// TwinCAT 3 PLC project Automation_App
// ProgramVersion: 3.1.4026.21
// libraries:
//   Tc2_MC2, * (Beckhoff Automation GmbH)
//   Tc2_Standard, * (Beckhoff Automation GmbH)
//   Tc2_System, * (Beckhoff Automation GmbH)
//   Tc2_Utilities, * (Beckhoff Automation GmbH)
//   Tc3_Module, * (Beckhoff Automation GmbH)
//   BASIC,3.31,OSCAT
// project tree:
//   GVLs/ GVL_VFD.TcGVL
//   / PlcTask.TcTTO
//   POUs/InputConveyor/ FB_InputConvBufferManagement.TcPOU, FB_InputConvVFD.TcPOU, FB_InputConvProperties.TcPOU, FB_InputConvMAIN.TcPOU, ST_InputConvData.TcDUT
//   POUs/ MAIN.TcPOU
//   POUs/OutputConveyor/ FB_OutputConvVFD.TcPOU, ST_OutputConvData.TcDUT, FB_OutputConvBufferManagement.TcPOU, FB_OutputConvMain.TcPOU, FB_OutputConvProperties.TcPOU
//   POUs/RobotInterface/ FB_RobotInterefaceMAIN.TcPOU
// real-time tasks:
//   TASK PlcTask: cycle T#1ms, priority 20, ADS port 350

CONFIGURATION Automation_App
    RESOURCE PLC ON TwinCAT3
        TASK PlcTask(INTERVAL := T#1ms, PRIORITY := 20);
        PROGRAM MAIN WITH PlcTask : MAIN;
    END_RESOURCE
END_CONFIGURATION

// ---- POUs/InputConveyor/ST_InputConvData.TcDUT
TYPE ST_InputConvData :
STRUCT
	id :INT; // Unique box identifier assigned on entry
	timeStampin :STRING; // Timestamp when box passed the entry (IN) sensor
	timeStamparrived:STRING; // Timestamp when box reached the exit (OUT) sensor
	timeStampout:STRING; // Timestamp when box cleared the exit (OUT) sensor
END_STRUCT
END_TYPE

// ---- POUs/OutputConveyor/ST_OutputConvData.TcDUT
TYPE ST_OutputConvData :
STRUCT
	id :INT; // Unique box identifier assigned when robot places the box
	timeStampin :STRING; // Timestamp when box entered the drop zone (IN sensor rising edge)
	timeStampout:STRING; // Timestamp when box left the conveyor (OUT sensor falling edge)
END_STRUCT
END_TYPE

// ---- GVLs/GVL_VFD.TcGVL
{attribute 'qualified_only'}
VAR_GLOBAL
	
// INPUT Conveyor----------------------
// Outputs from PLC to input conveyor VFD
	bInConvStop			AT%Q*:BOOL; // Stop command to input conveyor VFD
    bInConvRunFWD		AT%Q*:BOOL; // Run forward command to input conveyor VFD
	bInConvRunREV		AT%Q*:BOOL; // Run reverse command to input conveyor VFD
	bInConvJog			AT%Q*:BOOL; // Jog command to input conveyor VFD

// Inputs from input conveyor VFD to PLC
	bInputVFDSpeedReached	AT%I*:BOOL; // Speed-reached status from input conveyor VFD
	bInConvFault			AT%I*:BOOL; // Fault status from input conveyor VFD
	bInputVFDRunning		AT%I*:BOOL; // Running status from input conveyor VFD
	
// Inputs form Conveyor Sensors
	bInputConveyorINSensor	AT%I*:BOOL; // Entry photo sensor on input conveyor (box arriving)
	bInputConveyorOUTSensor AT%I*:BOOL; // Exit photo sensor on input conveyor (box at robot pickup position)

// OUTPUT CONVEYOR-----------------------
// Outputs from PLC to input conveyor VFD
	bOutConvStop		AT%Q*:BOOL; // Stop command to output conveyor VFD
    bOutConvRunFWD		AT%Q*:BOOL; // Run forward command to output conveyor VFD
	bOutConvRunREV		AT%Q*:BOOL; // Run reverse command to output conveyor VFD
	bOutConvJog			AT%Q*:BOOL; // Jog command to output conveyor VFD

// Inputs from input conveyor VFD to PLC
	bOutputVFDSpeedReached	AT%I*:BOOL; // Speed-reached status from output conveyor VFD
	bOutConvFault			AT%I*:BOOL; // Fault status from output conveyor VFD
	bOutputVFDRunning		AT%I*:BOOL; // Running status from output conveyor VFD
	
// Inputs form Conveyor Sensors
	bOutputConveyorINSensor		AT%I*:BOOL; // Entry photo sensor on output conveyor (robot drop zone)
	bOutputConveyorOUTSensor	AT%I*:BOOL; // Exit photo sensor on output conveyor (box leaving system)
END_VAR

// ---- POUs/MAIN.TcPOU
PROGRAM MAIN
VAR
    InputConveyor	:FB_InputConvMAIN;      // Input conveyor subsystem controller
	RobotInterface	:FB_RobotInterefaceMAIN; // Robot pick/place coordination
	OutputConveyor	:FB_OutputConvMAIN;     // Output conveyor subsystem controller

    bEnable		:BOOL; //PLC Logic Enable
	bInFeedtoConv :BOOL:= TRUE; // Allow external infeed system to feed boxes onto input conveyor
	rCyclePLC	:REAL:= 0.001; // PLC task cycle time in seconds (1 ms default)
	bSimulation :BOOL; // TRUE = run in simulation mode (no real hardware required)
	
END_VAR

InputConveyor(
	bEnable:= bEnable , 
	bInFeedtoConv:= bInFeedtoConv , 
	bRobotReadytoPick:= RobotInterface.bRobotReadyPickInputConv , 
	rCyclePLC:= rCyclePLC, 
	bSimulation:= bSimulation, 
	AllowInFeedtoInputConv=> , 
	AllowOutFeedtoRobot=> );

//RobotInterface
RobotInterface(
	bEnable := bEnable,
	bInputConvReady:= InputConveyor.AllowOutFeedtoRobot ,
	bOutputConvReady:= outputconveyor.AllowRobotPlace ,
	bRobotReadyPickInputConv=> ,
	bRobotReadyPlaceOutputConv=> );

//InputConveyor(
OutputConveyor(
	bEnable:= bEnable , 
	bRobotReadytoPlace:= RobotInterface.bRobotReadyPlaceOutputConv , 
	rCyclePLC:= rCyclePLC , 
	bSimulation:= bSimulation, 
	AllowRobotPlace=>);

END_PROGRAM

// ---- POUs/InputConveyor/FB_InputConvMAIN.TcPOU
FUNCTION_BLOCK FB_InputConvMAIN
VAR_INPUT
	bEnable			:BOOL; //PLC Logic Enable
	bInFeedtoConv 	:BOOL; //Outside signal from infeed system to conveyor - ready to recieve
	bRobotReadytoPick 	:BOOL; //Outside signal from robot - ready to recieve
	rCyclePLC			:REAL; // PLC task cycle time in seconds
	bSimulation :BOOL; // TRUE = VFD simulation active (no real drive)
	
END_VAR
VAR_OUTPUT
	AllowInFeedtoInputConv :BOOL; //Allow infeed of new boxes signal
	AllowOutFeedtoRobot :BOOL; //Ready to be picked up by robot signal
END_VAR
VAR
	//Function Blocks
	InputConvPropeties		:FB_InputConvProperties;
	InputConvVFD			:FB_InputConvVFD;
	InputConvBufferManger	:FB_InputConvBufferManagement;

	iMotorMaxSpeed			:INT; // Motor rated speed at 50 Hz [RPM]
	iConveyorVelocitycmd	:REAL; // Commanded belt velocity [m/s]
	rAccTime				:REAL; // Drive acceleration time [s]
	rDecTime				:REAL; // Drive deceleration time [s]

	//Belt linear vel tranformation
	iGearboxReduction	:INT := 1; // Gearbox reduction ratio (motor to pulley shaft)
	rPullyDiameter		:REAL; // Drive pulley diameter [m]
	
	//Conveyor propeties 
	rConvLength :REAL; //Conveyor Length in m (Distance between sensors)
	rBoxLen	:REAL; //Box size length in m
	rMinGap	:REAL; //Allowable min gap between boxes in m
	
END_VAR



InputConvBufferManger(
	bEnable:= bEnable , 
	bInSensor:= GVL_VFD.bInputConveyorINSensor, 
	bOutSensor:= GVL_VFD.bInputConveyorOUTSensor ,
	bReadytoRecieve:= bInFeedtoConv, 
	rConvLength:= rConvLength , 
	rBoxLen:= rBoxLen , 
	rMinGap:= rMinGap , 
	bRobotReady:= bRobotReadytoPick);

AllowInFeedtoInputConv := InputConvBufferManger.bAllowIn;
AllowOutFeedtoRobot := InputConvBufferManger.bAllowOut;
	
InputConvPropeties(
	GearboxReduction:= iGearboxReduction , 
	PullyDiameter:= rPullyDiameter , 
	ConveyorVelocitycmd:= iConveyorVelocitycmd  , 
	MotorMaxSpeed:= iMotorMaxSpeed,
	bBufferFull:= InputConvBufferManger.bFull);

IF bSimulation THEN 

	InputConvVFD(
		bStop:= GVL_VFD.bInConvStop, 
		bRunFWR:= GVL_VFD.bInConvRunFWD, 
		bRunREV:= GVL_VFD.bInConvRunREV , 
		bJog:= GVL_VFD.bInConvJog , 
		iVoltage:= InputConvPropeties.AnalogOut_V,
		iVoltageMax:= 10,
		rAccTime:= rAccTime , 
		rDecTime:= rDecTime,
		iMotorMaxSpeed:= iMotorMaxSpeed,
		ConveyorVelocityMax:= InputConvPropeties.ConveyorVelocityMax);
		
END_IF

GVL_VFD.bInputVFDSpeedReached	:= InputConvVFD.bSpeedReached;
GVL_VFD.bInputVFDRunning		:= InputConvVFD.bRunning;
//GVL_VFD.bInConvFault	:= ;

END_FUNCTION_BLOCK

// ---- POUs/InputConveyor/FB_InputConvProperties.TcPOU
FUNCTION_BLOCK FB_InputConvProperties
VAR_INPUT 
	bEnable				:BOOL; // PLC Logic Enable
	GearboxReduction 	:INT; // Gearbox reduction ratio (motor to pulley shaft)
	PullyDiameter		:REAL; //m
	ConveyorVelocitycmd	:REAL; //m/s
	MotorMaxSpeed		:INT; //RPM at 50 Hz (ASSUMPTION)
	bBufferFull			:BOOL; // Forces motor speed to zero when the conveyor buffer is full
	
END_VAR

VAR_OUTPUT
	ConveyorVelocityMax  :REAL; // [m/s] at MotorMaxSpeed
    MotorRPM             :REAL; // [rpm]
    MotorHz              :REAL; // [Hz] 0..50
    AnalogOut_V          :REAL; // [V] 0..10
    AnalogOut_Raw     AT%Q*: INT;   // 0..32767
END_VAR

VAR
	HzMax 	:REAL :=50; // Maximum drive frequency [Hz]
    HzCmd	:REAL; // Calculated frequency command [Hz]
    Vin		:REAL; // Calculated analog output voltage [V]
    RawAnalog	:REAL; // Intermediate raw analog value before INT conversion
END_VAR

IF PullyDiameter = 0.0 OR MotorMaxSpeed = 0 OR GearboxReduction = 0 THEN
	ConveyorVelocityMax := 0;
ELSE
	ConveyorVelocityMax := (PullyDiameter*PI*(MotorMaxSpeed/GearboxReduction))/60; // m/s
END_IF

IF bBufferFull THEN
    MotorRPM := 0.0;	// forced stop
ELSIF (PullyDiameter > 0.0) AND (GearboxReduction > 0.0) THEN
    MotorRPM := (ConveyorVelocitycmd * 60.0 * GearboxReduction) / (LREAL_TO_REAL (PI) * PullyDiameter);	// RPM
ELSE
    MotorRPM := 0.0;	// invalid mechanics
END_IF;

// RPM -> Hz (0..50)
IF (MotorMaxSpeed <= 0.0) THEN
	HzCmd := 0.0;
ELSE
	HzCmd := (MotorRPM / MotorMaxSpeed) * HzMax;
END_IF

// Clamp Hz to 0..50
IF HzCmd < 0.0 THEN
	HzCmd := 0.0;
ELSIF HzCmd > HzMax THEN
	HzCmd := HzMax;
END_IF
MotorHz := HzCmd;

// Hz -> 0..10V (linear)
Vin := (HzCmd / HzMax) * 10.0;

// Clamp V to 0..10
IF Vin < 0.0 THEN
	Vin := 0.0;
ELSIF Vin > 10.0 THEN
	Vin := 10.0;
END_IF
AnalogOut_V := Vin;

// 0..10V -> 0..32767 counts
RawAnalog := (Vin / 10.0) * 32767.0;

// Clamp counts
IF RawAnalog < 0.0 THEN
	RawAnalog := 0.0;
ELSIF RawAnalog > 32767.0 THEN
	RawAnalog := 32767.0;
END_IF

AnalogOut_Raw := REAL_TO_INT(LREAL_TO_REAL(RawAnalog));

END_FUNCTION_BLOCK

// ---- POUs/InputConveyor/FB_InputConvVFD.TcPOU
//Generate commands to a drive.
FUNCTION_BLOCK FB_InputConvVFD

VAR_INPUT
	bStop				:BOOL; // Stop command - resets SRAMP and forces velocity to zero
    bRunFWR				:BOOL; // Run forward command
	bRunREV				:BOOL; // Run reverse command
	bJog		:BOOL; // Jog command (treated the same as forward run)
	iVoltage		:REAL; // Analog speed reference voltage [V]
	iVoltageMax		:REAL; // Maximum analog reference voltage [V] (typically 10 V)
    rAccTime		:REAL;      // Acc in seconds
    rDecTime		:REAL;      // DEC in seconds
	iMotorMaxSpeed	:REAL; // Motor rated speed at 50 Hz [RPM]
	ConveyorVelocityMax :REAL; // Maximum conveyor belt velocity at motor max speed [m/s]
	
END_VAR

VAR_OUTPUT
	bSpeedReached	:BOOL; // TRUE when drive output frequency matches the reference
	bFault			:BOOL; // Drive fault flag (not implemented in simulation)
	bRunning		:BOOL; // TRUE when drive is running with a positive frequency reference
	rDriveVelProfile	:REAL;   // Simulated Motor vel profile
	rDriveACCProfile	:REAL; // Simulated Motor acc profile
	
END_VAR

VAR
	DriveRun		:BOOL; // TRUE when exactly one direction command is active (XOR result)
    DriveRunFWR		:BOOL; // Internal forward run (RunFWR OR Jog)
    DriveRunREV		:BOOL; // Internal reverse run
    DriveHzRef		:REAL; // Target frequency reference [Hz], ±HzMax
	rAccRate		:REAL; // Acceleration rate [Hz/s]
    rDecRate		:REAL; // Deceleration rate [Hz/s] (negative value)
	rDirSign 		:REAL; // Direction sign: +1.0 forward, -1.0 reverse
	fbSRAMP :SRAMP; // OSCAT S-ramp function block for smooth velocity profiling
	HzMax :REAL := 50; // Maximum drive frequency [Hz]
	rRPMvel :REAL; // Simulated motor shaft speed [RPM]
	rLinearVel :REAL; // Simulated conveyor belt linear velocity [m/s]
	sStatus		:STRING(120);	// STATUS text

END_VAR

// Run command
DriveRunFWR := bRunFWR OR bJog;
DriveRunREV := bRunREV;

DriveRun := (DriveRunFWR XOR DriveRunREV);   // TRUE only if one is on

IF bRunFWR OR bJog THEN
    rDirSign := 1.0;
ELSIF bRunREV THEN
    rDirSign := -1.0;

END_IF;

//Voltage to Hz:
IF iVoltage <= 0.0  THEN //OR NOT DriveRun
    DriveHzRef := 0.0;
ELSIF iVoltage > iVoltageMax THEN
    DriveHzRef := HzMax;
ELSE
    DriveHzRef := (iVoltage / iVoltageMax) * HzMax;
END_IF;


IF ABS(DriveHzRef) < 0.001 AND rAccTime > 0 THEN
    rAccRate := (HzMax / 2) / rAccTime;
ELSIF rAccTime > 0.01 THEN
    rAccRate := DriveHzRef / rAccTime;
ELSE
    rAccRate := DriveHzRef * 10.0;
END_IF;

IF ABS(DriveHzRef) < 0.001 AND rDecTime > 0 THEN
    rDecRate := (HzMax / 2) / -rDecTime;
ELSIF rDecTime > 0.01 THEN
	rDecRate := DriveHzRef / -rDecTime;   // Hz/s
ELSE
	rDecRate := DriveHzRef * -10.0;      // Hz/s
END_IF;

// Determine target input
IF DriveRun THEN 
	DriveHzRef := DriveHzRef * rDirSign;
ELSE
	DriveHzRef := 0.0;
END_IF;

// SRAMP function to build velocity command
fbSRAMP(
    X           := DriveHzRef,
    A_UP        := rAccRate,
    A_DN        := rDecRate,
    VU_MAX      := rAccRate *1000,     // Jerk
    VD_MAX      := rDecRate *1000,     // Jerk
    LIMIT_HIGH  := HzMax,
    LIMIT_LOW   := -HzMax,
    RST         := bStop ,
    Y           => rDriveVelProfile,
    V           => rDriveACCProfile // Acctual Acc
);

rRPMvel := rDriveVelProfile/HzMax * iMotorMaxSpeed;
rLinearVel := rDriveVelProfile/HzMax * ConveyorVelocityMax;

//Status
bSpeedReached := (rDriveVelProfile = DriveHzRef AND DriveRun );
bRunning      := (DriveHzRef > 0 AND DriveRun);

//Drive Status (priority-based)
IF bStop THEN
    // SRAMP reset → forced stop
    sStatus := 'STOP';

ELSIF (DriveRunFWR AND DriveRunREV) THEN
    // Illegal command combination
    sStatus := 'Command Conflict: Run Farward and Reverse';

ELSIF NOT DriveRun THEN
    // No valid run command (XOR result = FALSE)
    sStatus := 'Stopped (No specific direction Run Command)';

ELSE
    // DriveRun = TRUE (exactly one direction active)

    IF bRunFWR OR bJog THEN
        sStatus := 'Running Farward';

    ELSIF bRunREV THEN
        sStatus := 'Running Reverse';

    END_IF
END_IF;

END_FUNCTION_BLOCK

// ---- POUs/InputConveyor/FB_InputConvBufferManagement.TcPOU
FUNCTION_BLOCK FB_InputConvBufferManagement
VAR_INPUT

	bEnable	:BOOL; // PLC Logic Enable
    bInSensor	:BOOL; // Photo sensors
    bOutSensor	:BOOL; // Photo sensors
	bReadytoRecieve	:BOOL; //Ready to recieve from Robot
	// iCapacity	:INT; // For real system 
	
	// Geometry 
    rConvLength	:REAL;	// usable buffer length for simulation (meters)
    rBoxLen		:REAL;	// box length along travel for simulation (meters)
    rMinGap		:REAL;	// minimum clear gap between boxes for simulation (meters)
	
	bInfeedReady :BOOL:= TRUE; // Infeed Handshake
    bRobotReady	:BOOL:= TRUE; // Robot Handshake

END_VAR

VAR CONSTANT
    iMax_Boxes_buffer	:INT := 500; //  Expected max capacity FIFO storage size
END_VAR

VAR_OUTPUT
    bFull		:BOOL;			// Buffer is full (box count >= effective capacity)
    bEmpty		:BOOL;			// Buffer is empty (no boxes on conveyor)
    bAllowIn	:BOOL;			//Allow infeeder 
    bAllowOut	:BOOL;			//Allow Robot Pick
	
END_VAR

VAR
	bEnableBuffer :BOOL; // Enables FIFO tracking (must be TRUE for box counting to run)
		
    rtIn		:R_TRIG;	// Rising edge detector for bInSensor
    rtOut		:R_TRIG;	// Rising edge detector for bOutSensor
	ftOutOff	:F_TRIG;	// falling edge detector for bOutSensor
	
	bReset		:BOOL := FALSE; // Reset count on rising edge
    rtReset		:R_TRIG;	// Ralling edge reset
	
	iCount       :INT;     // current box count
    bInEdge      :BOOL;    // IN rising edge
    bOutEdge     :BOOL;    // OUT rising edge
	
	// Time
    fbTime	:FB_LocalSystemTime := (bEnable := TRUE, dwCycle := 1); // Local system time FB for box timestamping
    sNow	:STRING; // Current timestamp as formatted string
	
	//stData : ST_Data;
	Inputlog     : ARRAY[1..iMax_Boxes_buffer] OF ST_InputConvData; // FIFO array storing box tracking records
	
	// FIFO storage
    iHead	:INT := 1; // Index of the oldest box (next to dequeue)
    iTail	:INT := 1; // Index of the next empty slot (where next box is enqueued)
    iQCount	:INT := 0; // Current number of boxes in the FIFO

	// ID generator
    iIdCounter : INT := 0; // Auto-incrementing box ID counter (wraps at 32767)

	// Effective capacity
    iEffCap  : INT; // Effective buffer capacity after clamping (>= 0)

	iCapacity	:INT; // Configured maximum number of boxes on conveyor
	// Capacity intermediates
    rPitch_m	:REAL; // Box pitch = box length + minimum gap [m]
    rCap		:REAL; // Float capacity before floor truncation
    iCapTmp		:INT; // Intermediate capacity before final clamping

	i :INT; // Loop index used during FIFO reset
	sStatus		:STRING(120);	// STATUS text
END_VAR

//Capacity calculation -  For simulation
// IF (rBoxLen <= 0.0) OR (rMinGap <= 0.0) OR (rConvLength <= 0.0) THEN
//     iCapTmp := 0;
// ELSE
//     rPitch_m := rBoxLen + rMinGap;
// 
//     IF rPitch_m <= 0.0 THEN
//         iCapTmp := 0;
//     ELSE
//         rCap := (rConvLength + rMinGap) / rPitch_m;
// 
//         // Round down
//         iCapTmp := REAL_TO_INT(FLOOR(rCap));
// 
//         IF iCapTmp < 0 THEN
// 			iCapTmp := 0; 
// 		END_IF
//     END_IF
// END_IF
// 
// iCapacity := iCapTmp;

// Clamp to FIFO storage
iEffCap := iCapacity;

IF iEffCap < 0 THEN
	iEffCap := 0;
END_IF

//Timestamps
fbTime();
IF fbTime.bValid THEN
    sNow := SYSTEMTIME_TO_STRING(fbTime.systemTime);
ELSE
    sNow := '';
END_IF

// Edge detection
rtIn(CLK := bInSensor);
rtOut(CLK := bOutSensor);
rtReset(CLK := bReset);
ftOutOff(CLK := bOutSensor);

bInEdge  := rtIn.Q;
bOutEdge := rtOut.Q;

//Reset
IF rtReset.Q THEN
	
    iHead := 1;
    iTail := 1;
    iQCount := 0;
	
    FOR i := 1 TO iMax_Boxes_buffer DO
        Inputlog[i].id := 0;
        Inputlog[i].timeStampIn := '';
        Inputlog[i].timeStampArrived := '';
        Inputlog[i].timeStampOut := '';
    END_FOR

END_IF
	
//FIFO tracking
IF bEnable AND bEnableBuffer AND fbTime.bValid THEN

    // 1) IN rising edge > Push (if not full)
    IF bInEdge THEN
        IF iQCount < iEffCap THEN

            // ID wrap protection
            IF iIdCounter >= 32767 THEN
				iIdCounter := 0; 
			END_IF
            iIdCounter := iIdCounter + 1;

            Inputlog[iTail].id := iIdCounter;
            Inputlog[iTail].timeStampIn := sNow;
            Inputlog[iTail].timeStampArrived := '';
            Inputlog[iTail].timeStampOut := '';

            // advance tail
            iTail := iTail + 1;
            IF iTail > iMax_Boxes_buffer THEN
				iTail := 1;
			END_IF

            iQCount := iQCount + 1;
        END_IF
    END_IF


    // 2) OUT rising edge > stamp ARRIVED on oldest (HEAD)
    IF bOutEdge THEN
        IF iQCount > 0 THEN
            Inputlog[iHead].timeStampArrived := sNow;
        END_IF
    END_IF


    // 3) OUT falling edge -> stamp OUT on oldest and POP
    IF ftOutOff.Q THEN
        IF iQCount > 0 THEN
            Inputlog[iHead].timeStampOut := sNow;

            // pop
            iHead := iHead + 1;
            IF iHead > iMax_Boxes_buffer THEN
				iHead := 1;
			END_IF

            iQCount := iQCount - 1;
        END_IF
    END_IF

END_IF


iCount := iQCount; //Number of boxes on conveyor
bEmpty := (iCount <= 0);
bFull  := (iEffCap > 0) AND (iCount >= iEffCap);

// Send infeeder allow signal
bAllowIn  := bEnable AND NOT bFull AND NOT bInSensor AND bInfeedReady AND bReadytoRecieve;

// Outfeed release allowed if buffer has boxes AND robot is ready AND out sensor is blocked
bAllowOut := bEnable AND NOT bEmpty AND bOutSensor AND bRobotReady;

// Status (priority-based)
IF NOT bEnable THEN
    sStatus := 'Input-Conveyor Buffer - Disabled';

	// Hard limit states
	ELSIF bFull THEN
		sStatus := 'Conveyor is Full: STOP';
	ELSIF bEmpty THEN
		sStatus := 'Conveyor is Empty';

	// Infeed path (not full, not empty)
	ELSIF NOT bAllowIn THEN
		// Give the most relevant reason
		IF bInSensor THEN
			sStatus := 'Infeed blocked: entry sensor occupied';
		ELSIF NOT bInfeedReady THEN
			sStatus := 'Infeed blocked: infeeder not ready';
		ELSIF NOT bReadytoRecieve THEN
			sStatus := 'Infeed blocked: buffer not ready to receive';
		ELSE
			sStatus := 'Infeed blocked';
		END_IF

	// Outfeed path
	ELSIF NOT bAllowOut THEN
		IF NOT bOutSensor THEN
			sStatus := 'Outfeed waiting: no box at out sensor';
		ELSIF NOT bRobotReady THEN
			sStatus := 'Outfeed waiting: robot not ready';
		ELSE
			sStatus := 'Outfeed blocked';
		END_IF
ELSE
    sStatus := 'Running: Infeed/Outfeed allowed';
END_IF

END_FUNCTION_BLOCK

// ---- POUs/RobotInterface/FB_RobotInterefaceMAIN.TcPOU
FUNCTION_BLOCK FB_RobotInterefaceMAIN
VAR_INPUT
	bEnable :BOOL; // PLC Logic Enable
	bInputConvReady :BOOL; // Signal from input conveyor: box is ready at robot pickup position
	bOutputConvReady :BOOL; // Signal from output conveyor: drop zone is clear
	
END_VAR

VAR_OUTPUT
	bRobotReadyPickInputConv :BOOL; // Permission to robot: OK to pick from input conveyor
	bRobotReadyPlaceOutputConv :BOOL; // Permission to robot: OK to place on output conveyor
	
END_VAR
VAR
	
END_VAR

IF bEnable THEN
	bRobotReadyPickInputConv := TRUE;
	bRobotReadyPlaceOutputConv := TRUE;
ELSE
	bRobotReadyPickInputConv := FALSE;
	bRobotReadyPlaceOutputConv := FALSE;
END_IF

END_FUNCTION_BLOCK

// ---- POUs/OutputConveyor/FB_OutputConvMain.TcPOU
FUNCTION_BLOCK FB_OutputConvMAIN
VAR_INPUT
	bEnable				:BOOL; //PLC Logic Enable
	bRobotReadytoPlace 	:BOOL; // Outside signal from robot: ready to place a box
	rCyclePLC			:REAL; // PLC task cycle time in seconds
	bSimulation			:BOOL; // TRUE = VFD simulation active (no real drive)
	
END_VAR
VAR_OUTPUT
	AllowRobotPlace :BOOL; //Ready to be picked up by robot signal
END_VAR
VAR
	//Function Blocks
	OutputConvPropeties		:FB_OutputConvProperties;
	OutputConvVFD			:FB_OutputConvVFD;
	OutputConvBufferManger	:FB_OutputConvBufferManagement;
//	HMIStates				:FB_HMIStates;
	
	iMotorMaxSpeed			:INT; // Motor rated speed at 50 Hz [RPM]
	iConveyorVelocitycmd	:REAL; // Commanded belt velocity [m/s]
	rAccTime				:REAL; // Drive acceleration time [s]
	rDecTime				:REAL; // Drive deceleration time [s]

	//Belt linear vel tranformation
	iGearboxReduction	:INT := 1; // Gearbox reduction ratio (motor to pulley shaft)
	rPullyDiameter		:REAL; // Drive pulley diameter [m]
	
END_VAR

OutputConvBufferManger(
	bEnable:= bEnable, 
	bInSensor:= GVL_VFD.bOutputConveyorINSensor, 
	bOutSensor:= GVL_VFD.bOutputConveyorOUTSensor, 
	bRobotReadytoPlace:= bRobotReadytoPlace,  
	bEmpty=> , 
	bAllowDrop=> );
	
AllowRobotPlace := OutputConvBufferManger.bAllowDrop;

OutputConvPropeties(
	bEnable:= bEnable , 
	GearboxReduction:= iGearboxReduction , 
	PullyDiameter:= rPullyDiameter, 
	ConveyorVelocitycmd:= iConveyorVelocitycmd, 
	MotorMaxSpeed:= iMotorMaxSpeed );
	
IF bSimulation THEN 

	OutputConvVFD(
		bStop:= GVL_VFD.bOutConvStop, 
		bRunFWR:= GVL_VFD.bOutConvRunFWD, 
		bRunREV:= GVL_VFD.bOutConvRunREV , 
		bJog:= GVL_VFD.bOutConvJog , 
		iVoltage:= OutputConvPropeties.AnalogOut_V,
		iVoltageMax:= 10,
		rAccTime:= rAccTime , 
		rDecTime:= rDecTime,
		iMotorMaxSpeed:= iMotorMaxSpeed,
		ConveyorVelocityMax:= OutputConvPropeties.ConveyorVelocityMax);
END_IF
GVL_VFD.bOutputVFDSpeedReached	:= OutputConvVFD.bSpeedReached;
GVL_VFD.bOutputVFDRunning	:= OutputConvVFD.bRunning;

END_FUNCTION_BLOCK

// ---- POUs/OutputConveyor/FB_OutputConvProperties.TcPOU
FUNCTION_BLOCK FB_OutputConvProperties
VAR_INPUT 
	bEnable				:BOOL; // PLC Logic Enable
	GearboxReduction 	:INT; // Gearbox reduction ratio (motor to pulley shaft)
	PullyDiameter		:REAL; //m
	ConveyorVelocitycmd	:REAL; //m/s
	MotorMaxSpeed		:INT; //RPM at 50 Hz (ASSUMPTION)
	
END_VAR

VAR_OUTPUT
	ConveyorVelocityMax	:REAL; // [m/s] at MotorMaxSpeed
    MotorRPM			:REAL; // [rpm]
    MotorHz             :REAL; // [Hz] 0..50
    AnalogOut_V         :REAL; // [V] 0..10
    AnalogOut_Raw		AT%Q*: INT;   // 0..32767
END_VAR

VAR
	HzMax 		:REAL := 50; // Maximum drive frequency [Hz]
    HzCmd		:REAL; // Calculated frequency command [Hz]
    Vin			:REAL; // Calculated analog output voltage [V]
    RawAnalog	:REAL; // Intermediate raw analog value before INT conversion
END_VAR

IF PullyDiameter = 0.0 OR MotorMaxSpeed = 0 OR GearboxReduction = 0 THEN
	ConveyorVelocityMax := 0;
ELSE
	ConveyorVelocityMax := (PullyDiameter*PI*(MotorMaxSpeed/GearboxReduction))/60; // m/s
END_IF

IF (PullyDiameter > 0.0) AND (GearboxReduction > 0.0) THEN
    MotorRPM := (ConveyorVelocitycmd * 60.0 * GearboxReduction) / (LREAL_TO_REAL (PI) * PullyDiameter);	// RPM
ELSE
    MotorRPM := 0.0;	// invalid mechanics
END_IF;

// RPM -> Hz (0..50)
IF (MotorMaxSpeed <= 0.0) THEN
	HzCmd := 0.0;
ELSE
	HzCmd := (MotorRPM / MotorMaxSpeed) * HzMax;
END_IF

// Clamp Hz to 0..50
IF HzCmd < 0.0 THEN
	HzCmd := 0.0;
ELSIF HzCmd > HzMax THEN
	HzCmd := HzMax;
END_IF
MotorHz := HzCmd;

// Hz -> 0..10V (linear)
Vin := (HzCmd / HzMax) * 10.0;

// Clamp V to 0..10
IF Vin < 0.0 THEN
	Vin := 0.0;
ELSIF Vin > 10.0 THEN
	Vin := 10.0;
END_IF
AnalogOut_V := Vin;

// 0..10V -> 0..32767 counts
RawAnalog := (Vin / 10.0) * 32767.0;

// Clamp counts
IF RawAnalog < 0.0 THEN
	RawAnalog := 0.0;
ELSIF RawAnalog > 32767.0 THEN
	RawAnalog := 32767.0;
END_IF

AnalogOut_Raw := REAL_TO_INT(LREAL_TO_REAL(RawAnalog));

END_FUNCTION_BLOCK

// ---- POUs/OutputConveyor/FB_OutputConvVFD.TcPOU
//Generate commands to a drive.
FUNCTION_BLOCK FB_OutputConvVFD

VAR_INPUT
	bStop				:BOOL; // Stop command - resets SRAMP and forces velocity to zero
    bRunFWR				:BOOL; // Run forward command
	bRunREV				:BOOL; // Run reverse command
	bJog		:BOOL; // Jog command (treated the same as forward run)
	iVoltage		:REAL; // Analog speed reference voltage [V]
	iVoltageMax		:REAL; // Maximum analog reference voltage [V] (typically 10 V)
    rAccTime		:REAL;      // Acc in seconds
    rDecTime		:REAL;      // DEC in seconds
	iMotorMaxSpeed :REAL; // Motor rated speed at 50 Hz [RPM]
	ConveyorVelocityMax :REAL; // Maximum conveyor belt velocity at motor max speed [m/s]
END_VAR

VAR_OUTPUT
	bSpeedReached	:BOOL; // TRUE when drive output frequency matches the reference
	bFault			:BOOL; // Drive fault flag (not implemented in simulation)
	bRunning		:BOOL; // TRUE when drive is running with a positive frequency reference
	rDriveVelProfile	:REAL;   // Simulated Motor vel profile
	rDriveACCProfile	:REAL; // Simulated Motor acc profile
	
END_VAR

VAR
	DriveRun		:BOOL; // TRUE when exactly one direction command is active (XOR result)
    DriveRunFWR		:BOOL; // Internal forward run (RunFWR OR Jog)
    DriveRunREV		:BOOL; // Internal reverse run
    DriveHzRef		:REAL; // Target frequency reference [Hz], ±HzMax
	rAccRate		:REAL; // Acceleration rate [Hz/s]
    rDecRate		:REAL; // Deceleration rate [Hz/s] (negative value)
	rDirSign 		:REAL; // Direction sign: +1.0 forward, -1.0 reverse
	fbSRAMP :SRAMP; // OSCAT S-ramp function block for smooth velocity profiling
	HzMax :REAL := 50; // Maximum drive frequency [Hz]
	rRPMvel :REAL; // Simulated motor shaft speed [RPM]
	rLinearVel :REAL; // Simulated conveyor belt linear velocity [m/s]
	sStatus		:STRING(120);	// STATUS text

END_VAR

// Run command
DriveRunFWR := bRunFWR OR bJog;
DriveRunREV := bRunREV;

DriveRun := (DriveRunFWR XOR DriveRunREV);   // TRUE only if one is on

IF bRunFWR OR bJog THEN
    rDirSign := 1.0;
ELSIF bRunREV THEN
    rDirSign := -1.0;

END_IF;

//Voltage to Hz:
IF iVoltage <= 0.0  THEN //OR NOT DriveRun
    DriveHzRef := 0.0;
ELSIF iVoltage > iVoltageMax THEN
    DriveHzRef := HzMax;
ELSE
    DriveHzRef := (iVoltage / iVoltageMax) * HzMax;
END_IF;


IF ABS(DriveHzRef) < 0.001 AND rAccTime > 0 THEN
    rAccRate := (HzMax / 2) / rAccTime;
ELSIF rAccTime > 0.01 THEN
    rAccRate := DriveHzRef / rAccTime;
ELSE
    rAccRate := DriveHzRef * 10.0;
END_IF;

IF ABS(DriveHzRef) < 0.001 AND rDecTime > 0 THEN
    rDecRate := (HzMax / 2) / -rDecTime;
ELSIF rDecTime > 0.01 THEN
	rDecRate := DriveHzRef / -rDecTime;   // Hz/s
ELSE
	rDecRate := DriveHzRef * -10.0;      // Hz/s
END_IF;

// Determine target input
IF DriveRun THEN 
	DriveHzRef := DriveHzRef * rDirSign;
ELSE
	DriveHzRef := 0.0;
END_IF;

// SRAMP function to build velocity command
fbSRAMP(
    X           := DriveHzRef,
    A_UP        := rAccRate,
    A_DN        := rDecRate,
    VU_MAX      := rAccRate *1000,     // Jerk
    VD_MAX      := rDecRate *1000,     // Jerk
    LIMIT_HIGH  := HzMax,
    LIMIT_LOW   := -HzMax,
    RST         := bStop ,
    Y           => rDriveVelProfile,
    V           => rDriveACCProfile // Acctual Acc
);
rRPMvel:= rDriveVelProfile/HzMax * iMotorMaxSpeed;
rLinearVel := rDriveVelProfile/HzMax * ConveyorVelocityMax;

//Status
bSpeedReached := (rDriveVelProfile = DriveHzRef AND DriveRun);
bRunning      := (DriveHzRef > 0 AND DriveRun);

//Drive Status (priority-based)
IF bStop THEN
    // SRAMP reset → forced stop
    sStatus := 'STOP';

ELSIF (DriveRunFWR AND DriveRunREV) THEN
    // Illegal command combination
    sStatus := 'Command Conflict: Run Farward and Reverse';

ELSIF NOT DriveRun THEN
    // No valid run command (XOR result = FALSE)
    sStatus := 'Stopped (No specific direction Run Command)';

ELSE
    // DriveRun = TRUE (exactly one direction active)

    IF bRunFWR OR bJog THEN
        sStatus := 'Running Farward';

    ELSIF bRunREV THEN
        sStatus := 'Running Reverse';

    END_IF
END_IF;

END_FUNCTION_BLOCK

// ---- POUs/OutputConveyor/FB_OutputConvBufferManagement.TcPOU
FUNCTION_BLOCK FB_OutputConvBufferManagement
VAR_INPUT
    bEnable					: BOOL;
    bInSensor				: BOOL; // Entry sensor at robot drop zone
    bOutSensor				: BOOL; // Exit sensor at discharge
    bRobotReadytoPlace		: BOOL; // robot permission from robot
	
END_VAR

VAR CONSTANT
    iMax_Boxes_buffer : INT := 500;
END_VAR

VAR_OUTPUT
    bEmpty      : BOOL;
    bAllowDrop  : BOOL;     // allow robot to place a new box (entry sensor must be OFF)
END_VAR

VAR
    bEnableBuffer :BOOL; // Enables FIFO tracking (must be TRUE for box counting to run)
	rtIn     : R_TRIG; // Rising edge detector for bInSensor (box enters drop zone)
    ftOutOff : F_TRIG; // Falling edge detector for bOutSensor (box exits conveyor)

	bReset	: BOOL := FALSE; // Rising edge triggers full FIFO and counter reset
	rtReset	: R_TRIG; // Rising edge detector for bReset

    // Time
    fbTime : FB_LocalSystemTime := (bEnable := TRUE, dwCycle := 1); // Local system time FB for box timestamping
    sNow   : STRING; // Current timestamp as formatted string

    // FIFO
    Outputlog    : ARRAY[1..iMax_Boxes_buffer] OF ST_OutputConvData; // FIFO array storing box tracking records
    iHead   : INT := 1; // Index of the oldest box (next to dequeue)
    iTail   : INT := 1; // Index of the next empty slot (where next box is enqueued)
    iQCount : INT := 0; // Current number of boxes in the FIFO

    // ID generator
    iIdCounter : INT := 0; // Auto-incrementing box ID counter (wraps at 32767)

    i : INT; // Loop index used during FIFO reset
    sStatus : STRING(120); // Status text for diagnostics
END_VAR

// Time
fbTime();
IF fbTime.bValid THEN
    sNow := SYSTEMTIME_TO_STRING(fbTime.systemTime);
ELSE
    sNow := '';
END_IF

// Edge detection
rtIn(CLK := bInSensor);
ftOutOff(CLK := bOutSensor);
rtReset(CLK := bReset);

// Reset
IF rtReset.Q THEN
    iHead := 1;
    iTail := 1;
    iQCount := 0;

    FOR i := 1 TO iMax_Boxes_buffer DO
        Outputlog[i].id := 0;
        Outputlog[i].timeStampIn := '';
        Outputlog[i].timeStampOut := '';
    END_FOR
END_IF


IF bEnable AND bEnableBuffer AND fbTime.bValid THEN

    // 1) Entry rising edge -> PUSH
    // (robot placed a box; entry sensor went ON)
    IF rtIn.Q THEN
        // Basic protection: don't exceed storage
        IF iQCount < iMax_Boxes_buffer THEN

            IF iIdCounter >= 32767 THEN 
				iIdCounter := 0; 
			END_IF
            iIdCounter := iIdCounter + 1;

            Outputlog[iTail].id := iIdCounter;
            Outputlog[iTail].timeStampIn := sNow;
            Outputlog[iTail].timeStampOut := '';

            iTail := iTail + 1;
            IF iTail > iMax_Boxes_buffer THEN
				iTail := 1; 
			END_IF

            iQCount := iQCount + 1;

        END_IF
    END_IF


    // 2) Exit falling edge -> POP
    // (box left conveyor; exit sensor went OFF)
    IF ftOutOff.Q THEN
        IF iQCount > 0 THEN
            Outputlog[iHead].timeStampOut := sNow;

            iHead := iHead + 1;
            IF iHead > iMax_Boxes_buffer THEN
 				iHead := 1; 
			END_IF

            iQCount := iQCount - 1;

        END_IF
    END_IF
END_IF

// States
bEmpty := (iQCount <= 0);

// AllowDrop condition: ONLY if entry sensor is NOT ON (free zone)
// plus permissives if you keep them
bAllowDrop := bEnable AND bRobotReadytoPlace AND (NOT bInSensor);


// Status (optional)
IF NOT bEnable THEN
    sStatus := 'Output buffer disabled';
ELSIF bAllowDrop THEN
    sStatus := 'Running: drop allowed (entry sensor clear)';
ELSE
    IF bInSensor THEN
        sStatus := 'Drop blocked: entry sensor occupied';
    ELSIF NOT bRobotReadytoPlace THEN
        sStatus := 'Drop blocked: Robot is not ready to place';
    ELSE
        sStatus := 'Drop blocked';
    END_IF
END_IF

END_FUNCTION_BLOCK
